TYPE ST_CANopenObject :
STRUCT
	nIndex 		: DWORD;
	nSubIndex 	: DWORD;
	nLength 	: DWORD;
END_STRUCT
END_TYPE

(* stored: Version 1.1.0.1, ProductVersion 3.1.0.25
   DUT ST_CANopenObject: Id {df42f89a-c89f-4ccf-9f19-8fd8c891891a} *)
